Staubli VAL3: setCoords.pgx

program setCoords(string inputMessage (dimensions=1), num sio_ID (dimensions=1))
  local bool isNumber[2]
  local bool isOK
  local num msgLength
  local string reply
  local pointRx sampleCoordPnt
  local num xMsgIndex
  local num yMsgIndex
begin
  //**************************************************
  // Method to set the coordinates of currentSamPosj (current sample position).
  // Messages take the form:
  //     setCoords:#X1#Y2
  // Coordinate system starts at 0 (e.g. X=0, Y=0 is first sample position)
  //**************************************************

  // To start with the function is assumed working and we print the input
  isOK=true
  putln("Setting magazine coordinates based on:")
  putln("   "+inputMessage)


  // Find the where the coordinates are being supplied
  xMsgIndex=find(inputMessage,"#X")
  yMsgIndex=find(inputMessage,"#Y")
  msgLength=len(inputMessage)

  // Extract the coords from the message and convert string to number
  toNum(mid(inputMessage,(yMsgIndex-(xMsgIndex+2)),(xMsgIndex+2)),coords[0],isNumber[0])
  toNum(mid(inputMessage,(msgLength-(yMsgIndex+2)),(yMsgIndex+2)),coords[1],isNumber[1])

  // Check conversion to number successful and print to screen
  isOK=isOK and isNumber[0] and isNumber[1]
  if isNumber[0]==false
    reply="setCoords:fail_'Invalid X'"
    put("Failed setting X. Found: ")
    putln(right(inputMessage,(yMsgIndex-(xMsgIndex+2))))
  elseIf isNumber[1]==false
    reply="setCoords:fail_'Invalid Y'"
    put("Failed setting Y. Found: ")
    putln(right(inputMessage,(msgLength-(yMsgIndex+2))))
  endIf

  // Assuming we got the numbers, now we create our new joint coordinate
  if isOK==true
    put("Coords: X=")
    put(coords[0])
    put(" Y=")
    putln(coords[1])
    sampleCoordPnt=appro(jointToPoint(flange,world,homePosition),{(coords[0])*-17.03,(coords[1])*-17,0,0,0,0})
    isOK=pointToJoint(flange,homePosition,sampleCoordPnt,currentSamPosJ)

    if isOK==false
      reply="setCoords:fail_'Could not convert position to joint'"
      putln("Failed converting position to joint")
    else
      reply="setCoords:done"
    endIf
  endIf

  taskCreate "sendStatus",10,sendStatus(reply,sio_ID)
  taskKill("setCoords")
end
